FUNCTION_BLOCK TcoSequenceNonAutoRestorableTest EXTENDS TcoCore._internals_TcoContext
VAR
	_callMyPlcInstance	:	BOOL := FALSE;
	_sequencer : _TcoSequence(THIS^, NO.Structure, eRestoreMode.None);
	_runPLCinstanceOnce : BOOL := FALSE;
	_runPLCinstanceCyclicaly : BOOL := FALSE;
	_stepID : INT := 32764;
	_enabled : BOOL;
	_stepDescription : STRING := 'Last step sequence message';	
	_runOneStep : BOOL;
	_runAllSteps : BOOL;
	_finishStep : BOOL;
	_restore : BOOL;
	_cycleCount : INT;
	_restoreCycleCount : INT;
	_init: BOOL;
END_VAR

IF _callMyPlcInstance THEN
	IF NOT _init THEN
		ContextOpen();	
		ContextClose();	
		_init := THIS^._rtc.IsValid;
	END_IF
	
	IF _restore THEN
		ContextOpen();	
		THIS^._sequencer.Restore();	
		_restoreCycleCount := _restoreCycleCount + 1;
		_restore := FALSE;
		ContextClose();	
		RETURN;
	END_IF
	
	IF _runPLCinstanceOnce AND NOT _runPLCinstanceCyclicaly THEN
		ContextOpen();	
		THIS^.PLCinstanceRun(_stepID , _enabled, _stepDescription);
		_cycleCount := _cycleCount + 1;
		_runPLCinstanceOnce := FALSE;
		ContextClose();	
	END_IF
	
	IF _runPLCinstanceCyclicaly AND NOT _runPLCinstanceOnce THEN
		ContextOpen();	
		THIS^.PLCinstanceRun(_stepID , _enabled, _stepDescription);
		_cycleCount := _cycleCount + 1;
		ContextClose();	
	END_IF
END_IF;

{attribute 'TcRpcEnable'}
METHOD ChildHasAutoRestoreEnabled : BOOL;
ChildHasAutoRestoreEnabled := _sequencer.ChildHasAutoRestoreEnabled();
END_METHOD

{attribute 'TcRpcEnable'}
METHOD ChildIsAutoRestorable : BOOL;
ChildIsAutoRestorable := _sequencer.ChildIsAutoRestorable();
END_METHOD

{attribute 'TcRpcEnable'}
METHOD CleanupPointers
_sequencer.CleanupPointers();
END_METHOD

{attribute 'TcRpcEnable'}
METHOD ClearNumberOfSteps
_sequencer.ClearNumberOfSteps();
END_METHOD

{attribute 'TcRpcEnable'}
METHOD PROTECTED ContextClose
SUPER^._Close();
END_METHOD

{attribute 'TcRpcEnable'}
METHOD ContextOpen
SUPER^._Open();
END_METHOD

{attribute 'TcRpcEnable'}
METHOD GetChildState : INT
GetChildState := _sequencer.GetChildState();
END_METHOD

{attribute 'TcRpcEnable'}
METHOD GetCurrentStepOrder : UINT
GetCurrentStepOrder := _sequencer._currentStep.Order;
END_METHOD

{attribute 'TcRpcEnable'}
METHOD GetNumberOfStepsInSequence : UINT
GetNumberOfStepsInSequence := _sequencer._numberOfStepsInSequence;
END_METHOD

{attribute 'TcRpcEnable'}
METHOD GetOrderOfTheCurrentlyEvaluatedStep : UINT
GetOrderOfTheCurrentlyEvaluatedStep := _sequencer._theOrderOfTheCurrentlyEvaluatedStep;
END_METHOD

{attribute 'TcRpcEnable'}
METHOD GetOrderOfTheCurrentlyExecutedStep : UINT
GetOrderOfTheCurrentlyExecutedStep := _sequencer._theOrderOfTheCurrentlyExecutedStep;
END_METHOD

{attribute 'TcRpcEnable'}
METHOD GetPreviousNumberOfStepsInSequence : UINT
GetPreviousNumberOfStepsInSequence := _sequencer._previousNumberOfStepsInSequence;
END_METHOD

{attribute 'TcRpcEnable'}
METHOD GetRequestStepCycle : UINT
GetRequestStepCycle := _sequencer.RequestStepCycle;
END_METHOD

{attribute 'TcRpcEnable'}
METHOD GetSequencerErrorId : INT
GetSequencerErrorId := _sequencer.GetSequencerErrorId();
END_METHOD

{attribute 'TcRpcEnable'}
METHOD GetTextOfTheMostImportantMessage : STRING(254)
GetTextOfTheMostImportantMessage := THIS^._sequencer.GetTextOfTheMostImportantMessage();
END_METHOD

{attribute 'TcRpcEnable'}
METHOD HasAutoRestoreEnabled : BOOL;
HasAutoRestoreEnabled := _sequencer.HasAutoRestoreEnabled();
END_METHOD

{attribute 'TcRpcEnable'}
METHOD IsAutoRestorable : BOOL;
IsAutoRestorable := _sequencer.IsAutoRestorable();
END_METHOD

{attribute 'TcRpcEnable'}
METHOD IsFirstStepEntry : BOOL
IsFirstStepEntry := THIS^._sequencer.IsFirstStepEntry();
END_METHOD

METHOD PROTECTED  Main
END_METHOD

{attribute 'TcRpcEnable'}
METHOD PLCinstanceRun
VAR_INPUT
	inStepId			:	UINT;
	inEnabled			:	BOOL;
	inStepDescription	:	STRING(254);	
END_VAR
THIS^._sequencer.SetTestParams(	_runOneStep , _runAllSteps , _finishStep , inStepId , inEnabled , inStepDescription);

THIS^._sequencer._RunExecutionSubstitute();
END_METHOD

{attribute 'TcRpcEnable'}
METHOD RequestStep
VAR_INPUT
	inRequestedStepId : INT;
END_VAR
_sequencer._RequestStep(inRequestedStepId);
END_METHOD

{attribute 'TcRpcEnable'}
METHOD Restore
_sequencer.Restore();
END_METHOD

{attribute 'TcRpcEnable'}
METHOD SequenceComplete
_sequencer._SequenceComplete();
END_METHOD

{attribute 'TcRpcEnable'}
METHOD SequencerClose
THIS^._sequencer.SequencerClose();
END_METHOD

{attribute 'TcRpcEnable'}
METHOD SequencerHasError : BOOL
SequencerHasError := _sequencer.SequencerHasError();
END_METHOD

{attribute 'TcRpcEnable'}
METHOD SequencerOpen
THIS^._sequencer.SequencerOpen();
END_METHOD

{attribute 'TcRpcEnable'}
METHOD SetChildState
VAR_INPUT
	inState			:	INT;
END_VAR
_sequencer.SetChildState(inState);
END_METHOD

{attribute 'TcRpcEnable'}
METHOD SetCurrentStep
VAR_INPUT
	inStepID 			:	INT;
	inStepDescription	:	STRING(254);
END_VAR
_sequencer.SetCurrentStep(inStepID := inStepID, inStepDescription := inStepDescription);
END_METHOD

{attribute 'TcRpcEnable'}
METHOD SetCurrentStepToErrorState : BOOL
SetCurrentStepToErrorState := _sequencer.SetCurrentStepToErrorState();
END_METHOD

{attribute 'TcRpcEnable'}
METHOD SetCyclicMode : BOOL
SetCyclicMode := _sequencer.SetCyclicMode();
END_METHOD

{attribute 'TcRpcEnable'}
METHOD SetInvalidMode : BOOL
SetInvalidMode := _sequencer.SetInvalidMode();
END_METHOD

{attribute 'TcRpcEnable'}
METHOD SetNumberOfSteps : UINT
VAR_INPUT
	inNumberOfSteps :UINT;
END_VAR
_sequencer.SetNumberOfSteps(inNumberOfSteps);
SetNumberOfSteps := _sequencer._numberOfStepsInSequence;
END_METHOD

{attribute 'TcRpcEnable'}
METHOD SetRequestStepCycle : UINT
VAR_INPUT
	Value : UINT;
END_VAR
_sequencer.RequestStepCycle := Value;

SetRequestStepCycle := _sequencer.RequestStepCycle;
END_METHOD

{attribute 'TcRpcEnable'}
METHOD SetSequenceAsChecked : BOOL
VAR_INPUT
END_VAR
_sequencer.SetSequenceAsChecked();
END_METHOD

{attribute 'TcRpcEnable'}
METHOD SetSequenceAsNotChecked : BOOL
VAR_INPUT
END_VAR
_sequencer.SetSequenceAsNotChecked();
END_METHOD

{attribute 'TcRpcEnable'}
METHOD SetStepMode : BOOL
SetStepMode := _sequencer.SetStepMode();
END_METHOD

{attribute 'TcRpcEnable'}
METHOD Step : BOOL
VAR_INPUT
	inStepId			:	INT;
	inEnabled			:	BOOL;
	inStepDescription	:	STRING(254);		
END_VAR
Step := _sequencer._Step(inStepID := inStepId, inEnabled := inEnabled, inStepDescription := inStepDescription);
END_METHOD

{attribute 'TcRpcEnable'}
METHOD StepBackward
_sequencer._StepBackward();
END_METHOD

{attribute 'TcRpcEnable'}
METHOD StepCompleteWhen 
VAR_INPUT
	inCondition : BOOL;
END_VAR
_sequencer._StepCompleteWhen(inCondition);
END_METHOD

{attribute 'TcRpcEnable'}
METHOD StepForward
_sequencer._StepForward();
END_METHOD

{attribute 'TcRpcEnable'}
METHOD StepIn
_sequencer._StepIn();
END_METHOD

{attribute 'TcRpcEnable'}
METHOD UpdateCurrentStepDetails
VAR_INPUT
END_VAR
_sequencer.UpdateCurrentStepDetails();
END_METHOD

END_FUNCTION_BLOCK

(* stored: Version 1.1.0.1
   POU TcoSequenceNonAutoRestorableTest: Id {4700a902-5939-07ac-2134-79f0740da481}, SpecialFunc None
   Method ChildHasAutoRestoreEnabled: Id {39d48909-9c1d-0bc4-0c89-133d4335476c}
   Method ChildIsAutoRestorable: Id {52d5ca0f-3acc-05ba-1f29-492320087bc7}
   Method CleanupPointers: Id {5aaea55e-f572-0ffd-3664-e22f46cea930}
   Method ClearNumberOfSteps: Id {8bf3ccd8-1e00-0c59-2ba0-16c02978027c}
   Method ContextClose: Id {0ec730aa-8769-0826-3fb3-7ae08f553525}
   Method ContextOpen: Id {a5518d9e-0b13-00a8-330a-6cf5a787fe4c}
   Method GetChildState: Id {cb387d2a-c356-0576-23c7-00e60c3997e7}
   Method GetCurrentStepOrder: Id {7d1e2f82-7130-0224-322d-9c7c8a02228a}
   Method GetNumberOfStepsInSequence: Id {d2b71612-212e-088b-3989-fb56d19d091f}
   Method GetOrderOfTheCurrentlyEvaluatedStep: Id {0ff3eac9-61be-0889-3c44-cdbc273612a2}
   Method GetOrderOfTheCurrentlyExecutedStep: Id {8837826e-8dce-0d5b-3352-b7ec04168b9c}
   Method GetPreviousNumberOfStepsInSequence: Id {9c25a0d7-86db-01c0-385f-b17472a1be81}
   Method GetRequestStepCycle: Id {458fab61-54b9-02f2-24ea-fe2f93bb847d}
   Method GetSequencerErrorId: Id {366246d2-d0b0-097f-1321-cbe11b07ea42}
   Method GetTextOfTheMostImportantMessage: Id {501cfa33-4c43-0e0e-314f-569676c991bb}
   Method HasAutoRestoreEnabled: Id {cd5735bb-76c5-0744-0333-ddb3d44e92d1}
   Method IsAutoRestorable: Id {7fca43bb-96e0-0d99-08ac-dde08ec0706e}
   Method IsFirstStepEntry: Id {5d7a4526-e20f-05c5-0207-8171f89459c2}
   Method Main: Id {097e469b-677b-0bc7-11e5-e73aad27486d}
   Method PLCinstanceRun: Id {bf122f78-1269-0566-1da5-0a3cbaee719e}
   Method RequestStep: Id {ecc5a3e2-08c3-0322-3f5b-4bea34f974a6}
   Method Restore: Id {f4b0be62-691c-020c-31c1-9b4269917a1c}
   Method SequenceComplete: Id {22f095e9-45fe-00c8-2c25-d44ed91de335}
   Method SequencerClose: Id {19b4cfbc-8369-0cd5-1a96-19035ba16a40}
   Method SequencerHasError: Id {26a9d35e-d5d1-06ff-3e51-6650daeb1116}
   Method SequencerOpen: Id {2313c40e-d3a0-0c76-2ef5-0ab65c71abe5}
   Method SetChildState: Id {be6677c7-c97d-0ebb-2ef2-4279c295b787}
   Method SetCurrentStep: Id {8490471d-4e07-0b8d-197c-d95454d2c7aa}
   Method SetCurrentStepToErrorState: Id {05ec49d2-3972-0bd0-3d62-51969824ca79}
   Method SetCyclicMode: Id {1d9f4d47-1492-0909-3d81-12ea22da9a71}
   Method SetInvalidMode: Id {639dd581-8d52-0908-2a9f-d5d338a18dc2}
   Method SetNumberOfSteps: Id {fda15102-b5f9-02cd-3982-acd536a1b81c}
   Method SetRequestStepCycle: Id {2a59b804-5c6a-0ba6-32db-b4e7a77cbeb1}
   Method SetSequenceAsChecked: Id {944b368d-dd02-07c2-03d5-16643954d6c7}
   Method SetSequenceAsNotChecked: Id {e171080e-0187-0ba1-3d19-0a36c21cd6c8}
   Method SetStepMode: Id {a011dea8-5986-0fe9-2fbd-f43e2f5e8138}
   Method Step: Id {57df138d-8151-0f7e-08f9-3c911af84970}
   Method StepBackward: Id {3b6e49c2-d8e6-0ee9-10cd-8832342d5771}
   Method StepCompleteWhen: Id {b783bd4b-dc05-0e02-09b1-c07970aa08d8}
   Method StepForward: Id {28d02942-45bf-0ed7-3a0e-a22f4a77a429}
   Method StepIn: Id {cc7b3349-5c7a-0c7b-3646-cd41b13eda20}
   Method UpdateCurrentStepDetails: Id {f3f0b5f0-6e0c-0b3b-1879-dd5f05271854} *)
